{attribute addProperty BoxType "AT2040-0250-0023"}
{attribute addProperty Id "A_0106_AT2026_5250_0019_AT2026_5250AT2026_C5E5984862678.25"}
{attribute addProperty CRC "720029618"}
{attribute addProperty SizeInBites "626"}
{attribute addProperty SizeInBytes "78.25"}
TYPE A_0038_AT2040_0250_0023_2AEAC7B2 EXTENDS AT2040_BA5A9548 :
STRUCT
	{attribute addProperty Name "A_0106_AT2026_5250_0019_AT2026_5250"}
	A_0106_AT2026_5250_0019_AT2026_5250 : AT2026_C5E59848;
END_STRUCT
END_TYPE

(* stored: Version 1.2.0.0, ProductVersion 3.1.4024.9
   DUT A_0038_AT2040_0250_0023_2AEAC7B2: Id {873f9792-f339-48bd-b920-444dd8c6a769} *)
